// TIA Portal V17 export
// export: Created 2025-03-13T10:30:47.0674212Z, ExportSetting WithDefaults, DisplayName Totally Integrated Automation Portal, DisplayVersion V17 Update 8, DisplayName TIA Portal Openness, DisplayVersion V17 Update 8, DisplayName TIA Portal Version Control Interface, DisplayVersion V17, DisplayName SINAMICS Startdrive Advanced, DisplayVersion V17 SP2, DisplayName SINAMICS Startdrive G110M, G120, G120C, G120D, G120P, G115D, DisplayVersion V17 SP2, DisplayName SINAMICS Startdrive G130, G150, S120, S150, SINAMICS MV, S210, DisplayVersion V17 SP2, DisplayName STEP 7 Professional, DisplayVersion V17 Update 8, DisplayName SINUMERIK ONE STEP 7 Toolbox, DisplayVersion V17 Update 12, DisplayName SINUMERIK 840D sl STEP 7 Toolbox, DisplayVersion V17 Update 12, DisplayName STEP 7 Safety, DisplayVersion V17 Update 6, DisplayName WinCC Advanced, DisplayVersion V17 Update 8
DATA_BLOCK "DB148_CLADDING_AXIS_C22"   // DB148
{ DB_Accessible_From_OPC_UA := 'FALSE' }
AUTHOR : ETXETAR
VERSION : 1.0
// stored: AutoNumber false, DBAccessibleFromOPCUA false, DBAccessibleFromWebserver true, InstanceOfName FB32_AXIS, InstanceOfType FB
"FB32_AXIS"
   // VAR_INPUT
   //    OPTIONS_0 : Byte;
   //    OPTIONS_1 : Byte;
   //    SAFETY_BYPASS : Bool;
   //    OPTIMIZATION_BYPASS : Bool;
   //    AX_ENABLE : Bool;
   //    TEST_STOP_BRAKE_TEST_AX_NUM : Bool;
   //    PARAMETER_SET_0 : Bool;
   //    PARAMETER_SET_1 : Bool;
   //    PARAMETER_SET_2 : Bool;
   //    PARAMETER_SET_3 : Bool;
   //    MOVE_AXIS : Bool;
   //    SAFE_ENABLED : Bool;
   //    FEED_HOLD_COND : Bool;
   //    AX_TORQUE_ENABLE : Bool;
   //    MPP_AXIS_SELECTED : Bool;
   //    HMI_AXIS_SELECTED : Bool;
   //    HMI_REQ_LINE : Bool;
   //    JOG_MINUS_REQ_NOT_FC18 : Bool;
   //    JOG_PLUS_REQ_NOT_FC18 : Bool;
   //    JOG_MINUS_REQ_FC18 : Bool;
   //    JOG_PLUS_REQ_FC18 : Bool;
   //    FC18_EXTERNAL_POS : Real;
   //    AUTO_RETURN_COMMAND : Bool;
   //    AUTO_ADVANCE_COMMAND : Bool;
   //    DELETE_DISTANCE_TO_GO : Bool;
   //    FEED_OVERRIDE : Byte;
   //    FEED_OVER_ACTIVE : Bool;
   //    READ_POS : DWord;
   //    UNIT_ALARM : UInt;
   //    STATION_ALARM : UInt;
   // END_VAR
   // VAR_OUTPUT
   //    MOTOR_ACTIVE : Bool;
   //    MOVE_AX : Bool;
   //    FEED_HOLD_CONDITIONS : Bool;
   //    ACTIVE_PARAMETER_SET : Byte;
   //    AX_NOT_REFERENCE_ALM : Bool;
   //    AX_B_NOT_IN_PST_180_90_ALM : Bool;
   //    MAST_SLAVE_MODE_NOT_ACTIV_ALM : Bool;
   //    AX_TORQUE_EXCEEDED_ALM : Bool;
   //    AXIS_POS : Real;
   //    HMI_MOTION_EXECUTABILITY_LEFT : Bool;
   //    HMI_MOTION_EXECUTABILITY_RIGHT : Bool;
   //    HMI_MOTION_END_POS_LEFT : Bool;
   //    HMI_MOTION_END_POS_RIGHT : Bool;
   //    HMI_MOTION_ACTIVE_LEFT : Bool;
   //    HMI_MOTION_ACTIVE_RIGHT : Bool;
   // END_VAR
   // VAR_IN_OUT
   //    AxisDB : "LBP_typeAxisX";
   // END_VAR
   // VAR RETAIN
   //    AXIS { S7_SetPoint := 'True'} : "AXIS";
   //    TIMER_PULSES_ENABLE { S7_SetPoint := 'True'} : TOF_TIME;
   //    SAFETY_POSITIONS { S7_SetPoint := 'True'} : "FB33_SAFETY_POSITIONS";
   // END_VAR
BEGIN
END_DATA_BLOCK
